SUBAPPLICATION Uebung_151 (* Impulszähler *)
  (* Standard: 61499-2; Description: Copyright (c) 2023 Meisterschulen am Ostbahnhof This program and the accompanying materials are made available under the terms of the Eclipse Public License 2.0 which is available at https://www.eclipse.org/legal/epl-2.0/ SPDX-License-Identifier: EPL-2.0 *)
  (* Version 1.0, 2023-10-23, Franz Höpfinger, Meisterschulen am Ostbahnhof *)
  PACKAGE Uebungen;
  IMPORT logiBUS::io::PI::logiBUS_PI::PulseInput_I8;
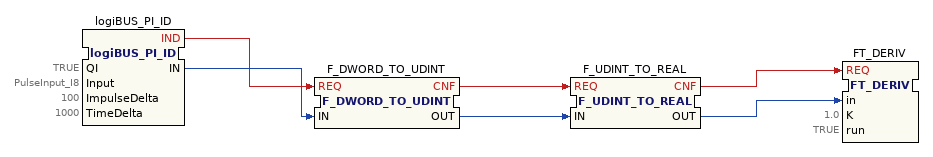
  FBS
    logiBUS_PI_ID : logiBUS::io::PI::logiBUS_PI_ID(QI := TRUE, Input := PulseInput_I8, ImpulseDelta := 100, TimeDelta := 1000);
    FT_DERIV : OSCAT::Basic::POUs::Engineering::Control::FT_DERIV(K := 1.0, run := TRUE);
    F_DWORD_TO_UDINT : iec61131::conversion::F_DWORD_TO_UDINT;
    F_UDINT_TO_REAL : iec61131::conversion::F_UDINT_TO_REAL;
  END_FBS
  EVENT_CONNECTIONS
    logiBUS_PI_ID.IND TO F_DWORD_TO_UDINT.REQ;
    F_DWORD_TO_UDINT.CNF TO F_UDINT_TO_REAL.REQ;
    F_UDINT_TO_REAL.CNF TO FT_DERIV.REQ;
  END_CONNECTIONS
  DATA_CONNECTIONS
    logiBUS_PI_ID.IN TO F_DWORD_TO_UDINT.IN;
    F_DWORD_TO_UDINT.OUT TO F_UDINT_TO_REAL.IN;
    F_UDINT_TO_REAL.OUT TO FT_DERIV.in;
  END_CONNECTIONS
END_SUBAPPLICATION
